FUNCTION F_CREATE_MESSAGE : BOOL
VAR_INPUT
END_VAR
VAR
END_VAR

END_FUNCTION

(* stored: Version 1.1.0.1
   POU F_CREATE_MESSAGE: Id {8220c5f4-cb2c-4878-8752-5687240a5aec}, SpecialFunc None *)
